// TIA Portal V17 export
// export: Created 2021-11-24T11:04:34.4918758Z, ExportSetting WithDefaults, DisplayName Totally Integrated Automation Portal, DisplayVersion V17, DisplayName TIA Portal Openness, DisplayVersion V17, DisplayName TIA Portal Version Control Interface, DisplayVersion V17, DisplayName SINAMICS Startdrive Advanced, DisplayVersion V17, DisplayName SINAMICS Startdrive G130, G150, S120, S150, SINAMICS MV, S210, DisplayVersion V17, DisplayName SINAMICS Startdrive G110M, G120, G120C, G120D, G120P, G115D, DisplayVersion V17, DisplayName STEP 7 Professional, DisplayVersion V17, DisplayName STEP 7 Safety, DisplayVersion V17, DisplayName WinCC Advanced / Unified PC, DisplayVersion V17
ORGANIZATION_BLOCK "Main"   // OB1, LAD, ProgramCycle
TITLE = "Main Program Sweep (Cycle)"
VERSION : 0.1
// stored: IsIECCheckEnabled false
   VAR_TEMP
      OB1_EV_CLASS : Byte;   // Bits 0-3 = 1 (Coming event), Bits 4-7 = 1 (Event class 1)
      OB1_SCAN_1 : Byte;   // 1 (Cold restart scan 1 of OB 1), 3 (Scan 2-n of OB 1)
      OB1_PRIORITY : Byte;   // Priority of OB Execution
      OB1_OB_NUMBR : Byte;   // 1 (Organization block 1, OB1)
      OB1_RESERVED_1 : Byte;   // Reserved for system
      OB1_RESERVED_2 : Byte;   // Reserved for system
      OB1_PREV_CYCLE : Int;   // Cycle time of previous OB1 scan (milliseconds)
      OB1_MIN_CYCLE : Int;   // Minimum cycle time of OB1 (milliseconds)
      OB1_MAX_CYCLE : Int;   // Maximum cycle time of OB1 (milliseconds)
      OB1_DATE_TIME : Date_And_Time;   // Date and time OB1 started
   END_VAR
BEGIN

REGION Network 1
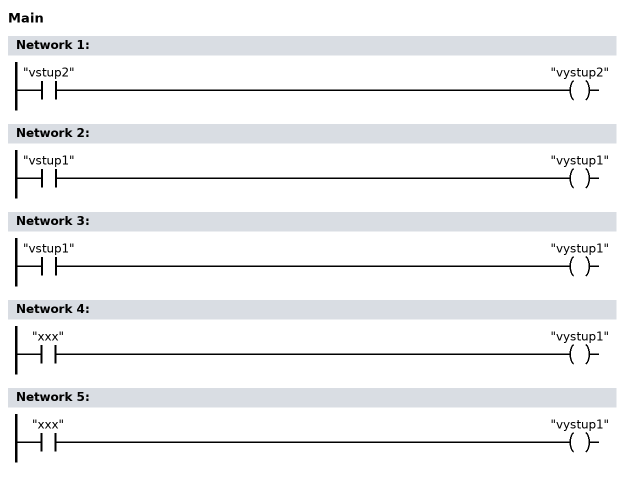
   RUNG wire#powerrail
      Contact( "vstup2" )
      Coil( "vystup2" )
   END_RUNG
   // the same network as SCL:
   "vystup2" := "vstup2";
END_REGION

REGION Network 2
   RUNG wire#powerrail
      Contact( "vstup1" )
      Coil( "vystup1" )
   END_RUNG
   // the same network as SCL:
   "vystup1" := "vstup1";
END_REGION

REGION Network 3
   RUNG wire#powerrail
      Contact( "vstup1" )
      Coil( "vystup1" )
   END_RUNG
   // the same network as SCL:
   "vystup1" := "vstup1";
END_REGION

REGION Network 4
   RUNG wire#powerrail
      Contact( "xxx" )
      Coil( "vystup1" )
   END_RUNG
   // the same network as SCL:
   "vystup1" := "xxx";
END_REGION

REGION Network 5
   RUNG wire#powerrail
      Contact( "xxx" )
      Coil( "vystup1" )
   END_RUNG
   // the same network as SCL:
   "vystup1" := "xxx";
END_REGION
END_ORGANIZATION_BLOCK
